(* PLC project Unnamed, Unknown Unnamed 1 *)
(* stored: creationDateTime 2013-01-29T14:01:00, modificationDateTime 2013-02-26T15:59:13 *)

FUNCTION_BLOCK EXIT_SIM
  VAR_INPUT
    TRIG : BOOL;
    EXIT_CODE : INT;
  END_VAR
  VAR
    TRIG0 : BOOL;
  END_VAR

IF TRIG AND NOT TRIG0 THEN
{{
    nsi_exit(GetFbVar(EXIT_CODE));
}}
END_IF;
TRIG0:=TRIG;

          
END_FUNCTION_BLOCK

FUNCTION_BLOCK SIM_PRINT
  VAR_INPUT
    TRIG : BOOL;
    MSG : STRING;
  END_VAR
  VAR
    TRIG0 : BOOL;
  END_VAR

IF TRIG AND NOT TRIG0 THEN
{{
    nsi_print_warning("%.*s\n", GetFbVar(MSG, .len),  (char*)GetFbVar(MSG, .body));
}}
END_IF;
TRIG0:=TRIG;

          
END_FUNCTION_BLOCK
